# EPICS autosave request: ADURL/urlApp/Db/URLDriver_settings.req
$(P)$(R)URL1
$(P)$(R)URL2
$(P)$(R)URL3
$(P)$(R)URL4
$(P)$(R)URL5
$(P)$(R)URL6
$(P)$(R)URL7
$(P)$(R)URL8
$(P)$(R)URL9
$(P)$(R)URL10
$(P)$(R)URLSelect.VAL
$(P)$(R)URLSelect.ZRST
$(P)$(R)URLSelect.ONST
$(P)$(R)URLSelect.TWST
$(P)$(R)URLSelect.THST
$(P)$(R)URLSelect.FRST
$(P)$(R)URLSelect.FVST
$(P)$(R)URLSelect.SXST
$(P)$(R)URLSelect.SVST
$(P)$(R)URLSelect.EIST
$(P)$(R)URLSelect.NIST
